TYPE ST_InputStationHSAdditionalDataGeneral :
STRUCT
	{attribute 'OPC.UA.DA.Description' := 'Dummy (for making struct visible on OPC UA'}
	{attribute 'TcIgnorePersistent'}
	Dummy						: BOOL;
END_STRUCT
END_TYPE

(* stored: Version 1.1.0.1, ProductVersion 3.1.4024.5
   DUT ST_InputStationHSAdditionalDataGeneral: Id {9755f085-f13b-4516-b1c6-e3eebf38af00} *)
